// TIA Portal V19 export
VAR_GLOBAL   // PLC tag table "TT - Feeding"
   iFeedingSenCilOut_k1 AT %I2.4 : Bool;
   iFeedingSenLoaded AT %I2.5 : Bool;
   "oFeedingVenCilOut_K+" AT %Q1.5 : Bool;
END_VAR
